TYPE ST_G120_Status :
(*
Version history:
Date		|	Version/Author 		|	Remark
----------------------------------------------------------------------------------------------------
09.02.18	|	2.000.016	PSA		|	Original Version.
									|	Siemens G120 drive structure
*)
STRUCT
	I								: ST_G120_IN;
	Q								: ST_G120_OUT;
END_STRUCT
END_TYPE

(* stored: Version 1.1.0.1, ProductVersion 3.1.4024.15
   DUT ST_G120_Status: Id {493ea123-23d7-4eb4-b166-2749a400cc14} *)
